(*	This FB is used for a single output solenoid 
	It uses the times to say when Extended/Retracted  	
	It starts assuming retracted and the output off.
*)
FUNCTION_BLOCK FB_A100 EXTENDS FB_ComponentBase IMPLEMENTS I_Cylinder
VAR
	//Output
	Output AT %Q* : BOOL;

	// Internal variables
	_ExtendRequest	: BOOL;
	_RetractRequest : BOOL;
	_Extended		: BOOL;
	_Retracted		: BOOL;
	_Extending		: BOOL;
	_Retracting		: BOOL;
	_ExtendTime		: LREAL := 1000; // Default time 1s
	_RetractTime	: LREAL := 1000; // Default time 1s

	// Timer for Extend/Retract
	Extend_TON	  : TON;
	Retract_TON	  : TON;
	Extend_RTRIG  : R_TRIG;
	Retract_RTRIG : R_TRIG;

	//HMI 
	Cylinder_HMI : ST_Cylinder_HMI;
END_VAR

METHOD PROTECTED CreateEvents
VAR_INPUT
END_VAR
SUPER^.CreateEvents();
END_METHOD

METHOD CyclicLogic
//One shot the requests
Extend_RTRIG(CLK := _ExtendRequest);
Retract_RTRIG(CLK := _RetractRequest);

//Handle Extend
IF Extend_RTRIG.Q THEN
	Output			:= TRUE;
	_Extending		:= TRUE;
	_Retracting		:= FALSE;
	_Retracted		:= FALSE;
	_RetractRequest := FALSE;
END_IF

//Handle Retract
IF Retract_RTRIG.Q THEN
	Output		   := FALSE;
	_Extending	   := FALSE;
	_Retracting	   := TRUE;
	_Extended	   := FALSE;
	_ExtendRequest := FALSE;
END_IF

//Handle the time to Extend/Retract
Extend_TON(IN := _Extending, PT := LREAL_TO_TIME(_ExtendTime));
Retract_TON(IN := _Retracting, PT := LREAL_TO_TIME(_RetractTime));
IF Extend_TON.Q THEN
	_Extended  := TRUE;
	_Extending := FALSE;
END_IF

IF Retract_TON.Q THEN
	_Retracted	:= TRUE;
	_Retracting := FALSE;
END_IF

SUPER^.CyclicLogic();
END_METHOD

METHOD Extend
_ExtendRequest	:= TRUE;
_RetractRequest := FALSE;
END_METHOD

PROPERTY Extended : BOOL
GET
Extended := _Extended;
END_GET
END_PROPERTY

PROPERTY ExtendTime : LREAL
GET
ExtendTime := _ExtendTime;
END_GET
SET
END_SET
END_PROPERTY

METHOD PROTECTED HMICommunication
VAR_INPUT
END_VAR
SUPER^.HMICommunication();

//Handle the requests to extend and retract
IF ComponentBase_HMI.Status.HMIControlAvailable THEN
	IF Cylinder_HMI.Command.Extend THEN
		Extend();
	ELSIF Cylinder_HMI.Command.Retract THEN
		Retract();
	END_IF
END_IF

//Update HMI status info
Cylinder_HMI.Status.Extended	:= _Extended;
Cylinder_HMI.Status.Extending	:= _Extending;
Cylinder_HMI.Status.Retracted	:= _Retracted;
Cylinder_HMI.Status.Retracting	:= _Retracting;
Cylinder_HMI.Config.ExtendTime	:= _ExtendTime;
Cylinder_HMI.Config.RetractTime := _RetractTime;
END_METHOD

//! @summary Basic component initialization logic
METHOD PROTECTED Initialize : BOOL;

//! @description This method is called by <c>CyclicLogic()</c> as required
//Set the cylinder to retracted
IF Output THEN
	_Extended  := TRUE;
	_Retracted := FALSE;
ELSE
	_Extended  := FALSE;
	_Retracted := TRUE;
END_IF

_Extending		:= FALSE;
_ExtendRequest	:= FALSE;
_Retracting		:= FALSE;
_RetractRequest := FALSE;

//Call base class Initialize
Initialize := SUPER^.Initialize();
END_METHOD

METHOD PROTECTED Monitoring
VAR_INPUT
END_VAR
_Busy	 := _Extending OR _Retracting;
_Error	 := FALSE;
_ErrorID := 0;
SUPER^.Monitoring();
END_METHOD

METHOD Retract
_ExtendRequest	:= FALSE;
_RetractRequest := TRUE;
END_METHOD

PROPERTY Retracted : BOOL
GET
Retracted := _Retracted;
END_GET
END_PROPERTY

PROPERTY RetractTime : LREAL
GET
RetractTime := _RetractTime;
END_GET
SET
_RetractTime := RetractTime;
END_SET
END_PROPERTY

END_FUNCTION_BLOCK

(* stored: Version 1.1.0.1, ProductVersion 3.1.4024.15
   POU FB_A100: Id {87fe144f-91bf-4463-866e-8a0be16a3639}, SpecialFunc None
   Folder I_ComponentBase: Id {270d4e9b-42c5-4718-80af-72f72ac26dae}
   Folder I_CyclicFB: Id {42980e1a-7cb7-48c4-8fdd-4239c59da53f}
   Folder I_Cylinder: Id {10f80a7f-327a-4f30-8855-e0c504bc3c85}
   Method CreateEvents: Id {ef9822f7-1819-4204-afad-c79a63fa0e6b}
   Method CyclicLogic: Id {da25161b-1e8e-4069-9a00-d8c255469adf}
   Method Extend: Id {2920103e-ded4-4315-8552-f17e6d19939b}
   Property Extended: Id {9d073ffe-27d2-44c4-8434-115418ff6a6b}
   Get Get: Id {e34b18d7-e84d-4d6a-ad83-767deaa59ee8}
   Property ExtendTime: Id {eef525ff-2de2-4293-a070-9330070bcc30}
   Get Get: Id {f4470ef6-f539-4f58-83f1-bfccc36021c9}
   Set Set: Id {bfdcce58-453d-4af5-9c8b-a488d521a299}
   Method HMICommunication: Id {99929a9e-4c33-4954-8e54-38c6f8dead3c}
   Method Initialize: Id {54d5e6b7-645f-4516-a459-924d0a334915}
   Method Monitoring: Id {700cde58-0ddd-4984-b1f6-d1258ad0e5e0}
   Method Retract: Id {9ac69fc0-6d91-4bed-ac3a-440904a4bc84}
   Property Retracted: Id {0ec39df9-2f65-436b-9475-723d6e4c5480}
   Get Get: Id {227cf16c-14d4-46ac-985f-80be1f8427bd}
   Property RetractTime: Id {3fcda7d3-15b1-48f7-aeb8-68111ca294e2}
   Get Get: Id {52f1fc21-4cf3-471c-9d75-529d30a9fae6}
   Set Set: Id {694bf6a4-6c4e-45e6-b3fc-8125ce67b3e2} *)
